// TIA Portal V20 export
TYPE "LBP_typePowerrideOutput"
TITLE = Powerride image / Image Powerride
// Output image of powerride / Image des sorties de Powerride
   STRUCT
      ledInfo : DWord;   // Led24..Led0
      scaleRed : Bool;   // when true, red scale LED is on / si vrai, la LED d'échelle rouge est allumée
      scaleGreen : Bool;   // when true, green scale LED is on / si vrai, la LED d'échelle verte est allumée
      scaleBlue : Bool;   // when true, blue scale LED ist on / si vrai, la LED d'échelle bleue est allumée
      buttonRed : Bool;   // when true, red push button LED is on / si vrai, la LED rouge du bouton-poussoir est allumée
      buttonGreen : Bool;   // when true, green push button LED is on / si vrai, la LED verte du bouton-poussoir est allumée
      buttonBlue : Bool;   // when true, blue push button LED is on / Si TRUE, la LED bleue du bouton-poussoir est allumée
      reserved46 : Bool;
      reserved47 : Bool;
      vibrationPattern : USInt;   // vibration pattern index to be used / indice du modèle de vibration à utiliser
   END_STRUCT;
END_TYPE
